PROGRAM MAIN
VAR
	nTest : INT := 0;
	sTest : STRING := 'Test';
	bTest : BOOL := TRUE;
	
END_VAR

END_PROGRAM

(* stored: Version 1.1.0.1
   POU MAIN: Id {e2307088-b17e-48c6-9faa-ec267c48a4c3}, SpecialFunc None *)
